Staubli VAL3: page.pgx

public program page(string& menuname[], num index)
// set all the page in french
begin
  //
  //  PAGE
  //
  //
  // PALLET PAGE
  if index>=10 and index<=19
    title("< Page Palette >")
  endIf
  // PALLET VIEW PAGE
  if index>=100 and index<=109
    title("< Page Vue Palette >")
  endIf
  switch index
    //
    // PALLET
    //
    // Integrator programmer
    case 10,11
      menuname="Vue Programmme,Edition Palette,,,Assitant,RAZ,Précédent,Suivant"
    break
    // On Cycle
    case 13,14
      menuname="Vue Programmme,Edition Palette,,,,RAZ,Précédent,Suivant"
    break
    // VIEW PALLET
    case 100,101,102,103,104,105
      menuname="RAZ tout,,,,,RAZ,Précédent,Suivant"
    break
  endSwitch
end
